SYSTEM test_AX
  (* Standard: 61499-1; Classification: Training; ApplicationDomain: Agriculture; Function: Learning how to use 4diac; Type: Test Type; Description: Copyright (c) 2023, 2025 HR Agrartechnik GmbH, Meisterschulen am Ostbahnhof This program and the accompanying materials are made available under the terms of the Eclipse Public License 2.0 which is available at https://www.eclipse.org/legal/epl-2.0/ SPDX-License-Identifier: EPL-2.0 https://www.logibus.tech/ Training Hier kann man über "Change Type" andere Ventilsteuerung_Uebung_001 usw auswählen, und so Übung für Übung vollziehen. Quellen: 1. Mit Musterlösungen: https://github.com/Meisterschulen-am-Ostbahnhof-Munchen/4diac_training1 2. Ohne Musterlösungen: https://github.com/Meisterschulen-am-Ostbahnhof-Munchen/4diac_training1_empty *)
  (* Version 1.0, 2025-09-28, Franz Höpfinger, HR Agrartechnik GmbH *)
  PACKAGE Training_AX;
  IMPORT logiBUS::stations::Computers::C_00;
  APPLICATION App_AX (* Default App for Everything *)
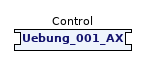
    SUBAPPS
      Control : Uebungen::Uebung_001_AX;
    END_SUBAPPS
  END_APPLICATION
  DEVICE FORTE_PC_AX : iec61499::system::FORTE_PC(MGR_ID := C_00 (* Device manager socket ID *))
    {SET_ATTRIBUTE(Profile, HOLOBLOC)}
    RESOURCE EMB_RES_AX : iec61499::system::EMB_RES
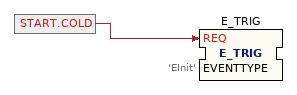
      FBS
        E_TRIG : iec61499::events::E_TRIG(EVENTTYPE := 'EInit');
      END_FBS
      EVENT_CONNECTIONS
        START.COLD TO E_TRIG.REQ;
      END_CONNECTIONS
    END_RESOURCE
  END_DEVICE
  MAPPINGS
    App_AX.Control ON FORTE_PC_AX.EMB_RES_AX;
  END_MAPPINGS
  SEGMENTS
    Ethernet : iec61499::system::Ethernet;
  END_SEGMENTS
  LINKS
    FORTE_PC_AX => Ethernet;
  END_LINKS
END_SYSTEM
